(* LS Electric XG5000 project: 제일교회 *)
(* PLC LSPLC *)
(* module base 0 slot 0: Cnet:XGL-C42A/B (Cnet 통신 모듈(RS-422/485, RS-422/485)) *)
(* module base 0 slot 1: 입력 모듈:XGI-D24A/B (DC 24V 입력, 32점 (전류소스 싱크공용/ 전류소스 입력)) *)
(* module base 0 slot 2: 입력 모듈:XGI-D21A (DC 24V 입력, 8점 (전류소스/싱크입력)) *)
(* module base 0 slot 3: 출력 모듈:XGQ-TR4A/B (트랜지스터 출력, 32점 (0.1A용, 싱크출력/소스출력)) *)

(* Comments on direct variables
%MX100	MAIN POWER PBL
%MX101	십자가 PBL
%MX102	강대상 위 천정 PBL
%MX103	강대석(좌) PBL
%MX104	무대조명(좌) PBL
%MX105	(미정) PBL
%MX106	본당벽체 간접 PBL
%MX107	복도(좌) PBL
%MX108	중벽체(반달 좌) PBL
%MX109	중벽체 간접(좌) PBL
%MX110	기둥간접(좌) PBL
%MX111	중앙천정 강대상 PBL
%MX112	중앙천정앞(50W전구색) PBL
%MX113	중앙천정좌 간접 PBL
%MX114	중앙천정우 간접 PBL
%MX115	중앙천정U(20W주광색) PBL
%MX116	중앙천정뒤(50W전구색) PBL
%MX117	강대석 (우) PBL
%MX118	무대조명(우) PBL
%MX119	(미정) PBL
%MX120	본당벽체 간접 PBL
%MX121	복도(우) PBL
%MX122	중벽채(반달 우) PBL
%MX123	중벽체 간접(우) PBL
%MX124	기둥간접(우) PBL
%MX125	2층 후미 PBL
%MX126	종탑 PBL
%MX127	LAMP TEST PBL
%MX128	BUZZER STOP PBL[SR]
%MX129	RESET PBL[SR]
%MX130	SPARE
%MX131	SPARE
%MX200	MAIN POWER IN
%MX201	십자가 IN
%MX202	강대상 위 천정 IN
%MX203	강대석(좌) IN
%MX204	무대조명(좌) IN
%MX205	(미정) IN
%MX206	본당벽체 간접 IN
%MX207	복도 IN
%MX208	중벽체(반달) IN
%MX209	중벽체 간접 IN
%MX210	기둥간접 IN
%MX211	중앙천정 강대상 IN
%MX212	중앙천정앞(50W전구색) IN
%MX213	중앙천정좌 간접 IN
%MX214	중앙천정우 간접 IN
%MX215	중앙천정U(20W주광색) IN
%MX216	중앙천정뒤(50W전구색) IN
%MX217	강대석 (우) IN
%MX218	무대조명(우) IN
%MX219	(미정) IN
%MX220	본당벽체 간접 IN
%MX221	복도 IN
%MX222	중벽채(반달) IN
%MX223	중벽체 간접 IN
%MX224	기둥간접 IN
%MX225	2층 후미 IN
%MX226	종탑 IN
%MX227	LAMP TEST IN
%MX228	BUZZER STOP IN
%MX229	RESET IN
%MX230	SPARE IN
%MX231	SPARE IN
%MX300	MAIN POWER OUT
%MX301	십자가 OUT
%MX302	강대상 위 천정 OUT
%MX303	강대석(좌) OUT
%MX304	무대조명(좌) OUT
%MX305	(미정) OUT
%MX306	본당벽체 간접 OUT
%MX307	복도 OUT
%MX308	중벽체(반달) OUT
%MX309	중벽체 간접 OUT
%MX310	기둥간접 OUT
%MX311	중앙천정 강대상 OUT
%MX312	중앙천정앞(50W전구색) OUT
%MX313	중앙천정좌 간접 OUT
%MX314	중앙천정우 간접 OUT
%MX315	중앙천정U(20W주광색) OUT
%MX316	중앙천정뒤(50W전구색) OUT
%MX317	강대석 (우) OUT
%MX318	무대조명(우) OUT
%MX319	(미정) OUT
%MX320	본당벽체 간접 OUT
%MX321	복도 OUT
%MX322	중벽채(반달) OUT
%MX323	중벽체 간접 OUT
%MX324	기둥간접 OUT
%MX325	2층 후미 OUT
%MX326	종탑 OUT
%MX327	LAMP TEST OUT
%MX328	BUZZER STOP OUT
%MX329	RESET OUT
%MX330	SPARE OUT
%MX331	SPARE OUT
%MX400	MAIN POWER REMOTE
%MX401	십자가 REMOTE
%MX402	강대상 위 천정 REMOTE
%MX403	강대석(좌) REMOTE
%MX404	무대조명(좌) REMOTE
%MX405	(미정) REMOTE
%MX406	본당벽체 간접 REMOTE
%MX407	복도 REMOTE
%MX408	중벽체(반달) REMOTE
%MX409	중벽체 간접 REMOTE
%MX410	기둥간접 REMOTE
%MX411	중앙천정 강대상
REMOTE
%MX412	중앙천정앞
50W전구색
REMOTE
%MX413	중앙천정좌 간접 REMOTE
%MX414	중앙천정우 간접 REMOTE
%MX415	중앙천정U(20W주광색) REMOTE
%MX416	중앙천정뒤(50W전구색) REMOTE
%MX417	강대석 (우) REMOTE
%MX418	무대조명(우) REMOTE
%MX419	(미정) REMOTE
%MX420	본당벽체 간접 REMOTE
%MX421	복도 REMOTE
%MX422	중벽채(반달) REMOTE
%MX423	중벽체 간접 REMOTE
%MX424	기둥간접 REMOTE
%MX425	2층 후미 REMOTE
%MX426	종탑 REMOTE
%MX427	LAMP TEST REMOTE
%MX428	BUZZER STOP REMOTE
%MX429	RESET REMOTE
%MX430	SPARE REMOTE
%MX431	SPARE REMOTE
%MX500	MAIN POWER LAMP
%MX501	십자가 LAMP
%MX502	강대상 위 천정 LAMP
%MX503	강대석(좌) LAMP
%MX504	무대조명(좌) LAMP
%MX505	(미정) LAMP
%MX506	본당벽체 간접 LAMP
%MX507	복도 LAMP
%MX508	중벽체(반달) LAMP
%MX509	중벽체 간접 LAMP
%MX510	기둥간접 LAMP
%MX511	중앙천정 강대상 LAMP
%MX512	중앙천정앞(50W전구색) LAMP
%MX513	중앙천정좌 간접 LAMP
%MX514	중앙천정우 간접 LAMP
%MX515	중앙천정U(20W주광색) LAMP
%MX516	중앙천정뒤(50W전구색) LAMP
%MX517	강대석 (우) LAMP
%MX518	무대조명(우) LAMP
%MX519	(미정) LAMP
%MX520	본당벽체 간접 LAMP
%MX521	복도 LAMP
%MX522	중벽채(반달) LAMP
%MX523	중벽체 간접 LAMP
%MX524	기둥간접 LAMP
%MX525	2층 후미 LAMP
%MX526	종탑 LAMP
%MX527	LAMP TEST LAMP
%MX528	BUZZER STOP LAMP
%MX529	RESET LAMP
%MX530	BUZZER
[REMOTE]
%MX531	SPARE LAMP
%MX911	Total Alarm
%MX1000	중앙1열 S/W
%MX1001	중앙2열 S/W
%MX1002	중앙3열 S/W
%MX1003	중앙4열 S/W
%MX1004	중앙5열 S/W
%MX1005	중앙6열 S/W
%MX1006	중앙7열 S/W
%MX1007	중앙8열 S/W
%MX1008	중앙9열 S/W
%MX1009	중앙10열 S/W
%MX1010	장로석 S/W
%MX1011	장로석 SPOT S/W
%MX1012	성가대 S/W
%MX1013	성가대 SPOT S/W
%MX1014	좌측통로 S/W
%MX1015	우측통로 S/W
%MX1016	후단1열 S/W
%MX1017	후단2열 S/W
%MX1018	후단3열 S/W
%MX1019	종탑 
S/W
%MX1020	중앙1열 M/C-a
%MX1021	중앙2열 M/C-a
%MX1022	중앙3열 M/C-a
%MX1023	중앙4열 M/C-a
%MX1024	중앙5열 M/C-a
%MX1025	중앙6열 M/C-a
%MX1026	중앙7열 M/C-a
%MX1027	중앙8열 M/C-a
%MX1028	중앙9열 M/C-a
%MX1029	중앙10열 M/C-a
%MX1030	장로석 M/C-a
%MX1031	장로석 SPOT M/C-a
%MX1200	중앙1열 LOGIC
%MX1201	중앙2열 LOGIC
%MX1202	중앙3열 LOGIC
%MX1203	중앙4열 LOGIC
%MX1204	중앙5열 LOGIC
%MX1205	중앙6열 LOGIC
%MX1206	중앙7열 LOGIC
%MX1207	중앙8열 LOGIC
%MX1208	중앙9열 LOGIC
%MX1209	중앙10열 LOGIC
%MX1210	장로석 LOGIC
%MX1211	장로석 SPOT-LOGIC
%MX1212	성가대 LOGIC
%MX1213	성가대 SPOT-LOGIC
%MX1214	좌측통로 LOGIC
%MX1215	우측통로 LOGIC
%MX1216	후단1열 LOGIC
%MX1217	후단2열 LOGIC
%MX1218	후단3열 LOGIC
%MX1219	종탑 
LOGIC
%MX1220	중앙1열 M/C-a
%MX1221	중앙2열 M/C-a
%MX1222	중앙3열 M/C-a
%MX1223	중앙4열 M/C-a
%MX1224	중앙5열 M/C-a
%MX1225	중앙6열 M/C-a
%MX1226	중앙7열 M/C-a
%MX1227	중앙8열 M/C-a
%MX1228	중앙9열 M/C-a
%MX1229	중앙10열 M/C-a
%MX1230	장로석 M/C-a
%MX1231	장로석 SPOT M/C-a
%MX2000	성가대 M/C-a
%MX2001	성가대 SPOT M/C-a
%MX2002	좌측통로 M/C-a
%MX2003	우측통로 M/C-a
%MX2004	후단1열 M/C-a
%MX2005	후단2열 M/C-a
%MX2006	후단3열 M/C-a
%MX2007	종탑 
M/C-a
%MX2200	성가대 M/C-a
%MX2201	성가대 SPOT M/C-a
%MX2202	좌측통로 M/C-a
%MX2203	우측통로 M/C-a
%MX2204	후단1열 M/C-a
%MX2205	후단2열 M/C-a
%MX2206	후단3열 M/C-a
%MW0	IN-COM0
%MW1	IN-COM1
%MW2	OUT-COM0
%MW3	OUT-COM1
%IX0.1.0	중앙1열 S/W
%IX0.1.1	중앙2열 S/W
%IX0.1.2	중앙3열 S/W
%IX0.1.3	중앙4열 S/W
%IX0.1.4	중앙5열 S/W
%IX0.1.5	중앙6열 S/W
%IX0.1.6	중앙7열 S/W
%IX0.1.7	중앙8열 S/W
%IX0.1.8	중앙9열 S/W
%IX0.1.9	중앙10열 S/W
%IX0.1.10	장로석 S/W
%IX0.1.11	장로석 SPOT S/W
%IX0.1.12	성가대 S/W
%IX0.1.13	성가대 SPOT S/W
%IX0.1.14	좌측통로 S/W
%IX0.1.15	우측통로 S/W
%IX0.1.16	후단1열 S/W
%IX0.1.17	후단2열 S/W
%IX0.1.18	후단3열 S/W
%IX0.1.19	종탑
%IX0.1.20	중앙1열 M/C-a
%IX0.1.21	중앙2열 M/C-a
%IX0.1.22	중앙3열 M/C-a
%IX0.1.23	중앙4열 M/C-a
%IX0.1.24	중앙5열 M/C-a
%IX0.1.25	중앙6열 M/C-a
%IX0.1.26	중앙7열 M/C-a
%IX0.1.27	중앙8열 M/C-a
%IX0.1.28	중앙9열 M/C-a
%IX0.1.29	중앙10열 M/C-a
%IX0.1.30	장로석 M/C-a
%IX0.1.31	장로석 SPOT M/C-a
%IX0.2.0	성가대 M/C-a
%IX0.2.1	성가대 SPOT M/C-a
%IX0.2.2	좌측통로 M/C-a
%IX0.2.3	우측통로 M/C-a
%IX0.2.4	후단1열 M/C-a
%IX0.2.5	후단2열 M/C-a
%IX0.2.6	후단3열 M/C-a
%IX0.2.7	종탑
M/C-a
%QX0.3.0	중앙1열
%QX0.3.1	중앙2열
%QX0.3.2	중앙3열
%QX0.3.3	중앙4열
%QX0.3.4	중앙5열
%QX0.3.5	중앙6열
%QX0.3.6	중앙7열
%QX0.3.7	중앙8열
%QX0.3.8	중앙9열
%QX0.3.9	중앙10열
%QX0.3.10	장로석
%QX0.3.11	장로석 SPOT
%QX0.3.12	성가대
%QX0.3.13	성가대 SPOT
%QX0.3.14	좌측통로
%QX0.3.15	우측통로
%QX0.3.16	후단1열
%QX0.3.17	후단2열
%QX0.3.18	후단3열
%QX0.3.19	종탑
%QX0.3.20	BUZZER
[MAIN]
*)

PROGRAM Communication (* task: 스캔 프로그램 *)
VAR
    IN_0_HIGH : BYTE;
    IN_0_LOW : BYTE;
    IN_1_HIGH : BYTE;
    IN_1_LOW : BYTE;
    OUT_0_HIGH : BYTE;
    OUT_0_LOW : BYTE;
END_VAR

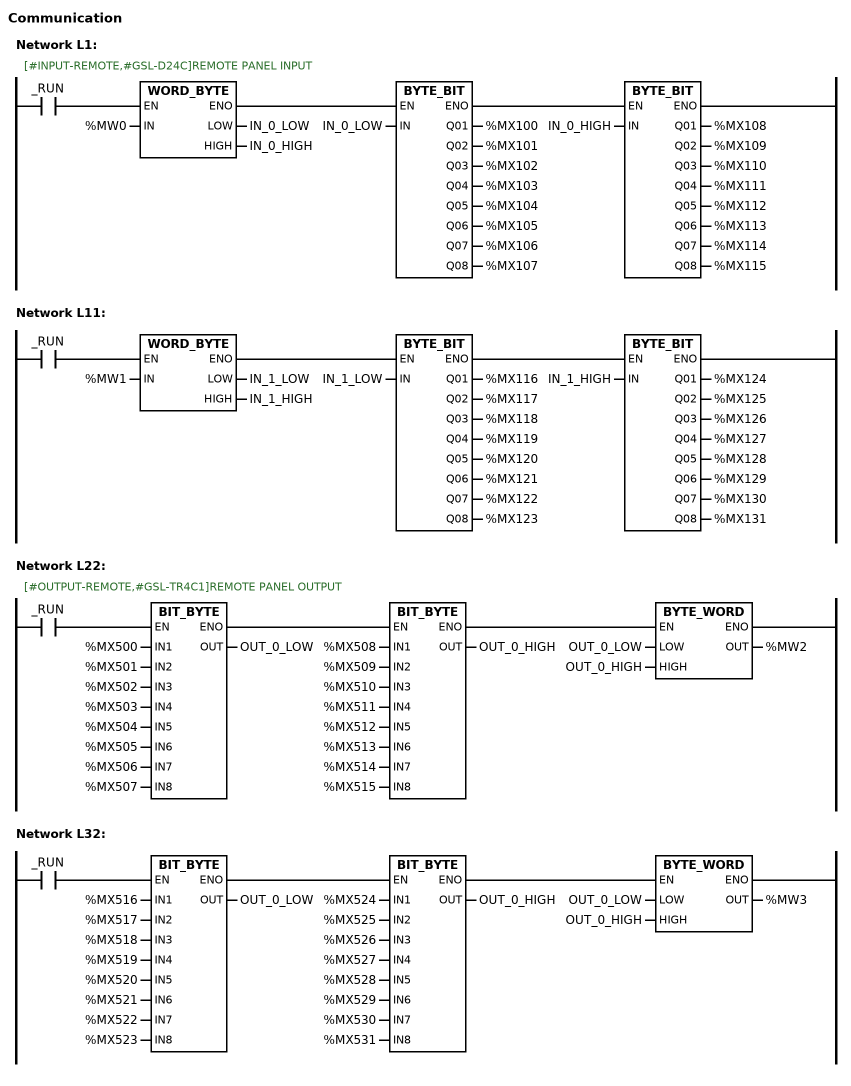
(* [#INPUT-REMOTE,#GSL-D24C]REMOTE PANEL INPUT *)
(* Rung L1 *)
IF _RUN THEN
    IN_0_LOW := WORD_BYTE(IN := %MW0, HIGH => IN_0_HIGH);
    %MX100 := BYTE_BIT(IN := IN_0_LOW, Q02 => %MX101, Q03 => %MX102, Q04 => %MX103, Q05 => %MX104, Q06 => %MX105, Q07 => %MX106, Q08 => %MX107);
    %MX108 := BYTE_BIT(IN := IN_0_HIGH, Q02 => %MX109, Q03 => %MX110, Q04 => %MX111, Q05 => %MX112, Q06 => %MX113, Q07 => %MX114, Q08 => %MX115);
END_IF;
(* Rung L11 *)
IF _RUN THEN
    IN_1_LOW := WORD_BYTE(IN := %MW1, HIGH => IN_1_HIGH);
    %MX116 := BYTE_BIT(IN := IN_1_LOW, Q02 => %MX117, Q03 => %MX118, Q04 => %MX119, Q05 => %MX120, Q06 => %MX121, Q07 => %MX122, Q08 => %MX123);
    %MX124 := BYTE_BIT(IN := IN_1_HIGH, Q02 => %MX125, Q03 => %MX126, Q04 => %MX127, Q05 => %MX128, Q06 => %MX129, Q07 => %MX130, Q08 => %MX131);
END_IF;
(* [#OUTPUT-REMOTE,#GSL-TR4C1]REMOTE PANEL OUTPUT *)
(* Rung L22 *)
IF _RUN THEN
    OUT_0_LOW := BIT_BYTE(%MX500, %MX501, %MX502, %MX503, %MX504, %MX505, %MX506, %MX507);
    OUT_0_HIGH := BIT_BYTE(%MX508, %MX509, %MX510, %MX511, %MX512, %MX513, %MX514, %MX515);
    %MW2 := BYTE_WORD(LOW := OUT_0_LOW, HIGH := OUT_0_HIGH);
END_IF;
(* Rung L32 *)
IF _RUN THEN
    OUT_0_LOW := BIT_BYTE(%MX516, %MX517, %MX518, %MX519, %MX520, %MX521, %MX522, %MX523);
    OUT_0_HIGH := BIT_BYTE(%MX524, %MX525, %MX526, %MX527, %MX528, %MX529, %MX530, %MX531);
    %MW3 := BYTE_WORD(LOW := OUT_0_LOW, HIGH := OUT_0_HIGH);
END_IF;
END_PROGRAM

PROGRAM Control-Remote (* task: 스캔 프로그램 *)
VAR
    FF0 : FF;
    FF1 : FF;
    FF10 : FF;
    FF11 : FF;
    FF12 : FF;
    FF13 : FF;
    FF14 : FF;
    FF15 : FF;
    FF16 : FF;
    FF17 : FF;
    FF18 : FF;
    FF19 : FF;
    FF2 : FF;
    FF20 : FF;
    FF21 : FF;
    FF22 : FF;
    FF23 : FF;
    FF24 : FF;
    FF25 : FF;
    FF26 : FF;
    FF27 : FF;
    FF28 : FF;
    FF29 : FF;
    FF3 : FF;
    FF30 : FF;
    FF31 : FF;
    FF4 : FF;
    FF5 : FF;
    FF6 : FF;
    FF7 : FF;
    FF8 : FF;
    FF9 : FF;
    INST : FF;
    INST1 : FF;
    IN_0_HIGH : BYTE;
    IN_0_LOW : BYTE;
    IN_1_HIGH : BYTE;
    IN_1_LOW : BYTE;
    off : BOOL;
END_VAR

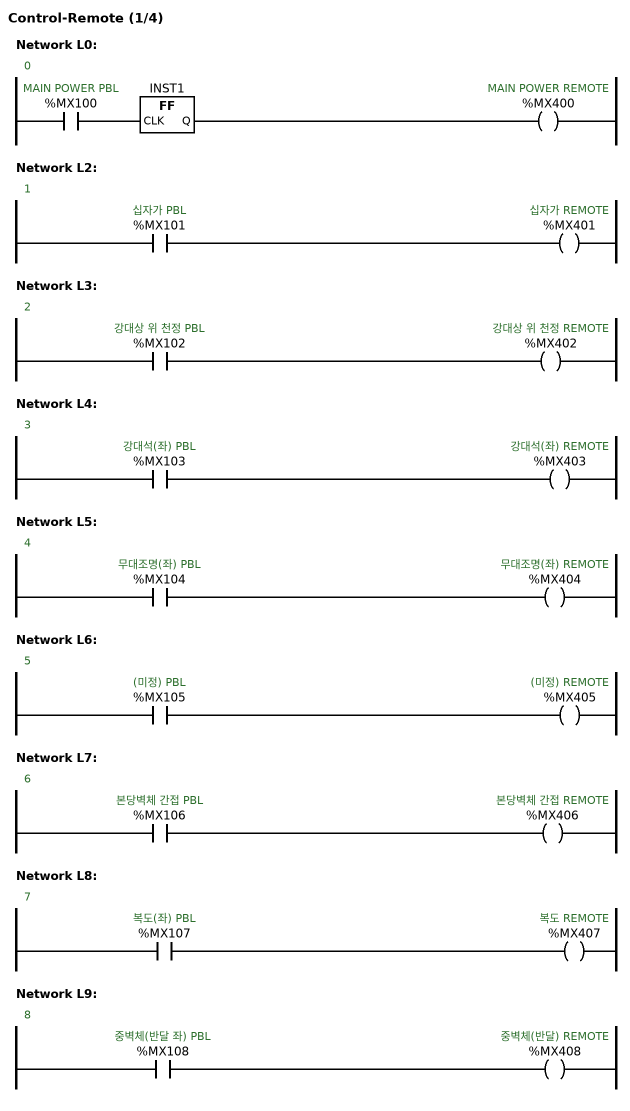
(* Rung L0 *)
INST1(CLK := %MX100);
%MX400 := INST1.Q;
(* 0 *)
(* Rung L2 *)
%MX401 := %MX101;
(* 1 *)
(* Rung L3 *)
%MX402 := %MX102;
(* 2 *)
(* Rung L4 *)
%MX403 := %MX103;
(* 3 *)
(* Rung L5 *)
%MX404 := %MX104;
(* 4 *)
(* Rung L6 *)
%MX405 := %MX105;
(* 5 *)
(* Rung L7 *)
%MX406 := %MX106;
(* 6 *)
(* Rung L8 *)
%MX407 := %MX107;
(* 7 *)
(* Rung L9 *)
%MX408 := %MX108;
(* 8 *)

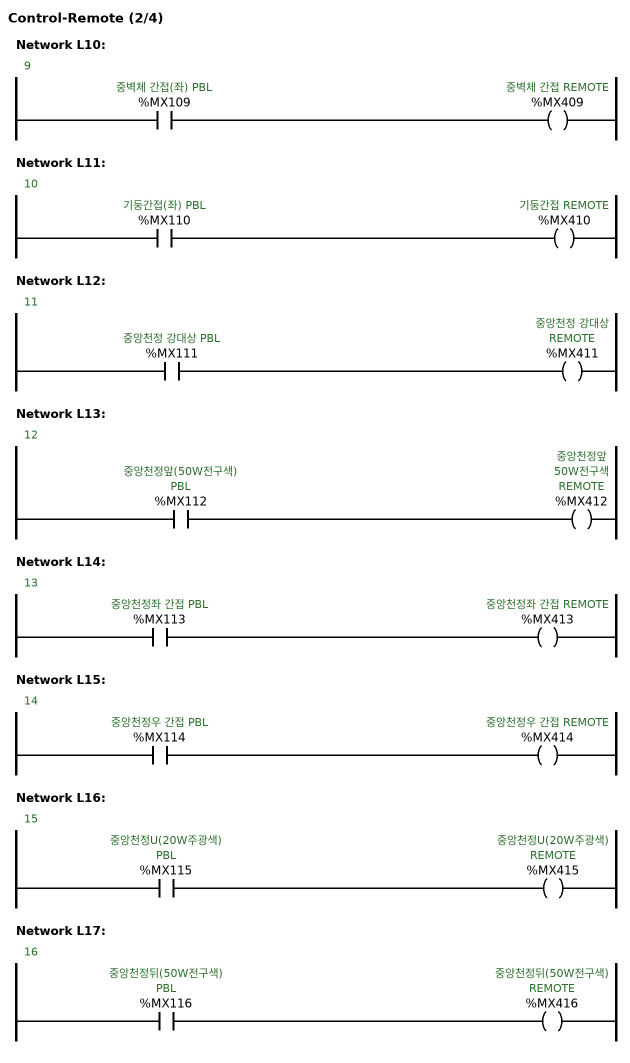
(* Rung L10 *)
%MX409 := %MX109;
(* 9 *)
(* Rung L11 *)
%MX410 := %MX110;
(* 10 *)
(* Rung L12 *)
%MX411 := %MX111;
(* 11 *)
(* Rung L13 *)
%MX412 := %MX112;
(* 12 *)
(* Rung L14 *)
%MX413 := %MX113;
(* 13 *)
(* Rung L15 *)
%MX414 := %MX114;
(* 14 *)
(* Rung L16 *)
%MX415 := %MX115;
(* 15 *)
(* Rung L17 *)
%MX416 := %MX116;
(* 16 *)

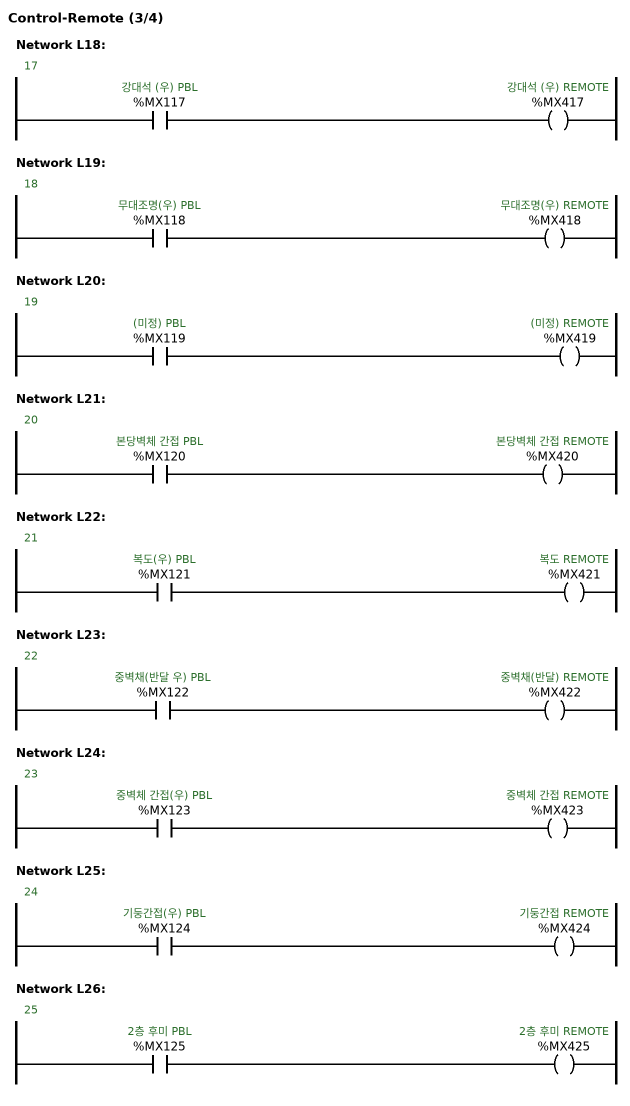
(* Rung L18 *)
%MX417 := %MX117;
(* 17 *)
(* Rung L19 *)
%MX418 := %MX118;
(* 18 *)
(* Rung L20 *)
%MX419 := %MX119;
(* 19 *)
(* Rung L21 *)
%MX420 := %MX120;
(* 20 *)
(* Rung L22 *)
%MX421 := %MX121;
(* 21 *)
(* Rung L23 *)
%MX422 := %MX122;
(* 22 *)
(* Rung L24 *)
%MX423 := %MX123;
(* 23 *)
(* Rung L25 *)
%MX424 := %MX124;
(* 24 *)
(* Rung L26 *)
%MX425 := %MX125;
(* 25 *)

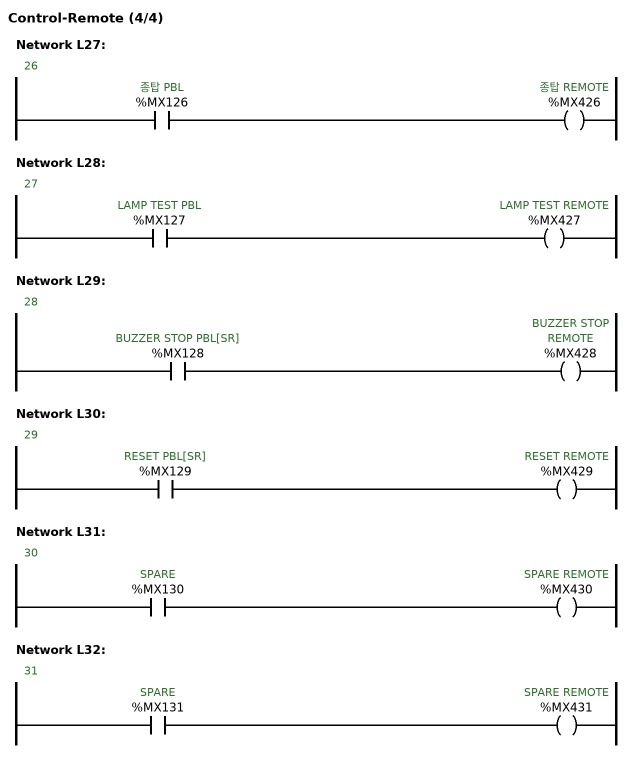
(* Rung L27 *)
%MX426 := %MX126;
(* 26 *)
(* Rung L28 *)
%MX427 := %MX127;
(* 27 *)
(* Rung L29 *)
%MX428 := %MX128;
(* 28 *)
(* Rung L30 *)
%MX429 := %MX129;
(* 29 *)
(* Rung L31 *)
%MX430 := %MX130;
(* 30 *)
(* Rung L32 *)
%MX431 := %MX131;
(* 31 *)
END_PROGRAM

PROGRAM Lamp-Remote (* task: 스캔 프로그램 *)
VAR
    INST : FF;
    INST1 : TMR_FLK;
    INST10 : TMR_FLK;
    INST2 : TMR_FLK;
    INST3 : TMR_FLK;
    INST4 : TMR_FLK;
    INST5 : TMR_FLK;
    INST6 : TMR_FLK;
    INST7 : TMR_FLK;
    INST8 : TMR_FLK;
    INST9 : TMR_FLK;
END_VAR

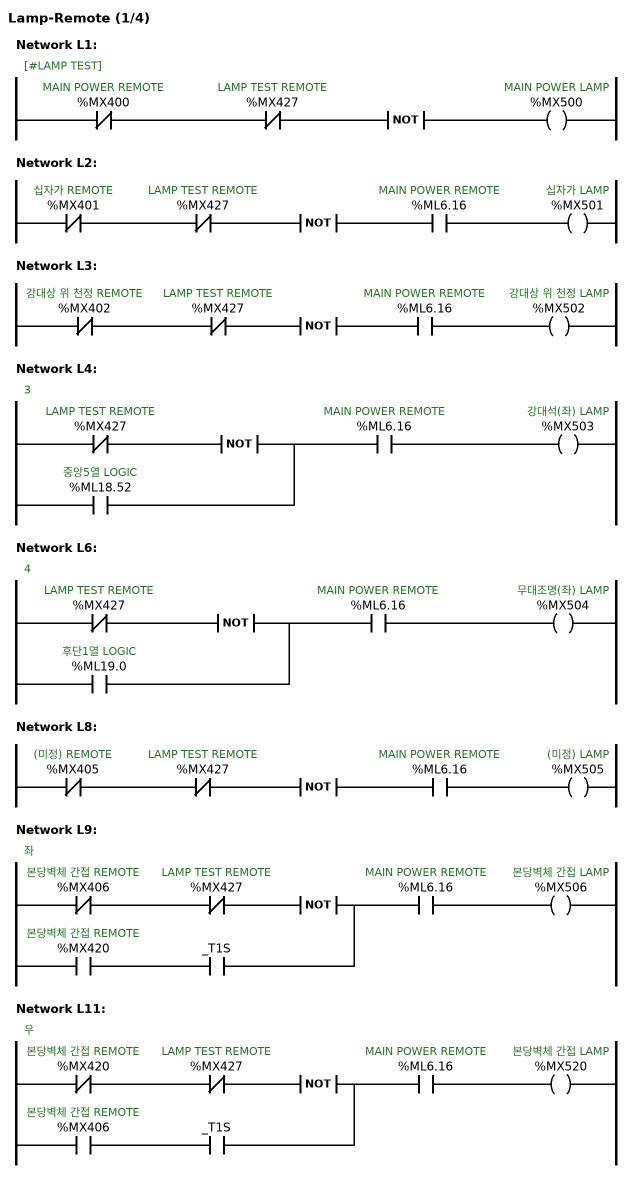
(* [#LAMP TEST] *)
(* Rung L1 *)
%MX500 := NOT (NOT %MX400 AND NOT %MX427);
(* Rung L2 *)
%MX501 := NOT (NOT %MX401 AND NOT %MX427) AND %ML6.16;
(* Rung L3 *)
%MX502 := NOT (NOT %MX402 AND NOT %MX427) AND %ML6.16;
(* Rung L4 *)
%MX503 := (%MX427 OR %ML18.52) AND %ML6.16;
(* 3 *)
(* Rung L6 *)
%MX504 := (%MX427 OR %ML19.0) AND %ML6.16;
(* 4 *)
(* Rung L8 *)
%MX505 := NOT (NOT %MX405 AND NOT %MX427) AND %ML6.16;
(* Rung L9 *)
%MX506 := (NOT (NOT %MX406 AND NOT %MX427) OR (%MX420 AND _T1S)) AND %ML6.16;
(* 좌 *)
(* Rung L11 *)
%MX520 := (NOT (NOT %MX420 AND NOT %MX427) OR (%MX406 AND _T1S)) AND %ML6.16;
(* 우 *)

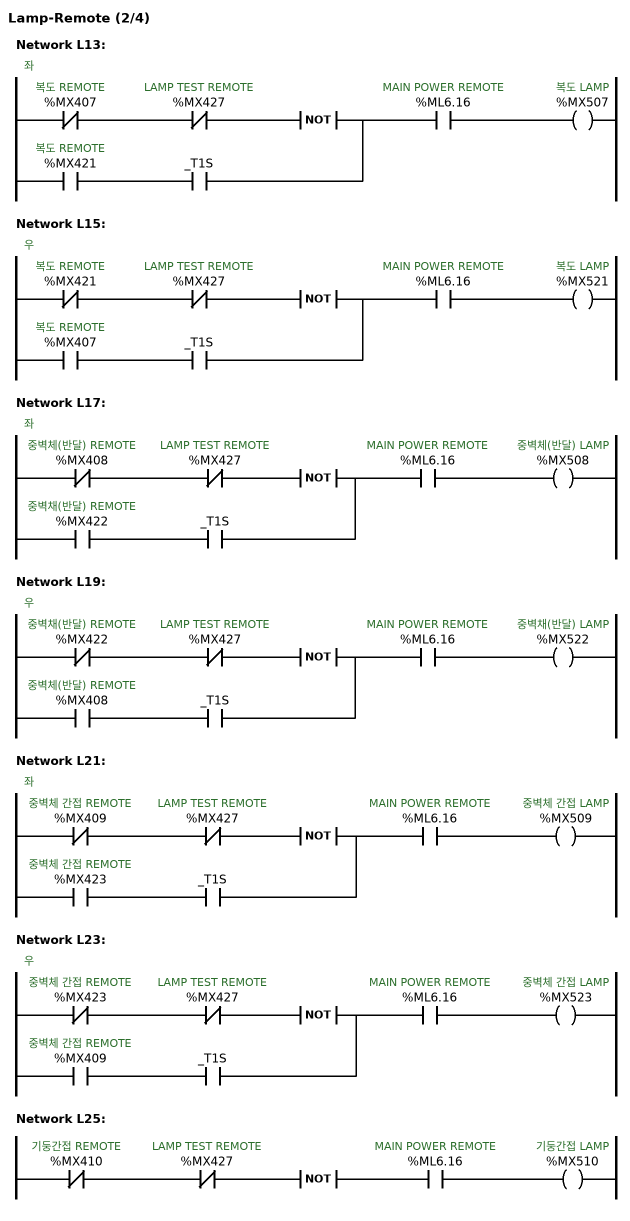
(* Rung L13 *)
%MX507 := (NOT (NOT %MX407 AND NOT %MX427) OR (%MX421 AND _T1S)) AND %ML6.16;
(* 좌 *)
(* Rung L15 *)
%MX521 := (NOT (NOT %MX421 AND NOT %MX427) OR (%MX407 AND _T1S)) AND %ML6.16;
(* 우 *)
(* Rung L17 *)
%MX508 := (NOT (NOT %MX408 AND NOT %MX427) OR (%MX422 AND _T1S)) AND %ML6.16;
(* 좌 *)
(* Rung L19 *)
%MX522 := (NOT (NOT %MX422 AND NOT %MX427) OR (%MX408 AND _T1S)) AND %ML6.16;
(* 우 *)
(* Rung L21 *)
%MX509 := (NOT (NOT %MX409 AND NOT %MX427) OR (%MX423 AND _T1S)) AND %ML6.16;
(* 좌 *)
(* Rung L23 *)
%MX523 := (NOT (NOT %MX423 AND NOT %MX427) OR (%MX409 AND _T1S)) AND %ML6.16;
(* 우 *)
(* Rung L25 *)
%MX510 := NOT (NOT %MX410 AND NOT %MX427) AND %ML6.16;

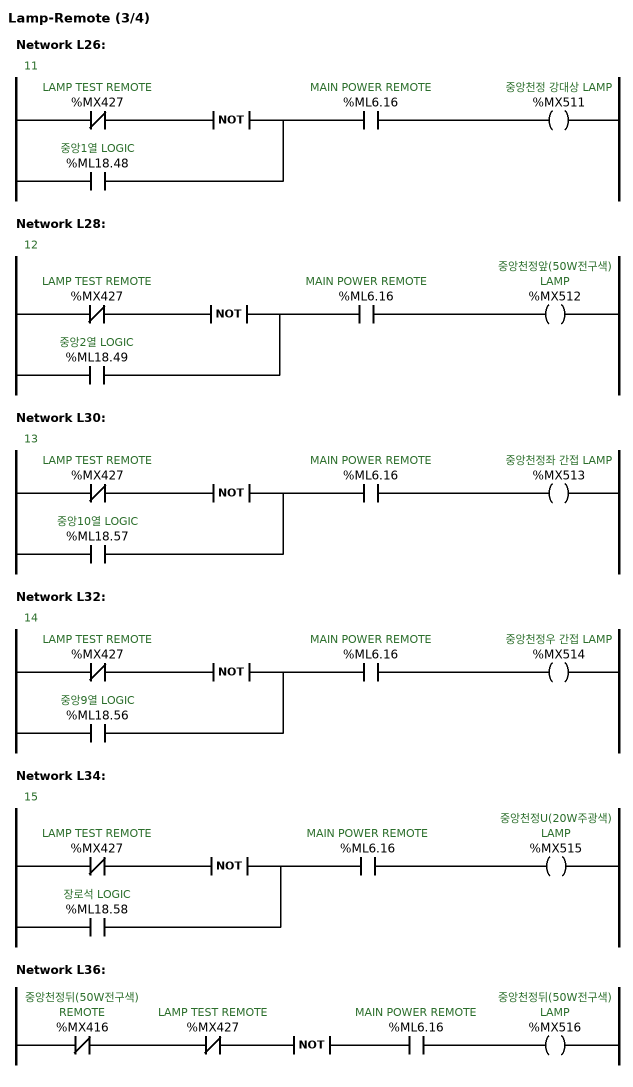
(* Rung L26 *)
%MX511 := (%MX427 OR %ML18.48) AND %ML6.16;
(* 11 *)
(* Rung L28 *)
%MX512 := (%MX427 OR %ML18.49) AND %ML6.16;
(* 12 *)
(* Rung L30 *)
%MX513 := (%MX427 OR %ML18.57) AND %ML6.16;
(* 13 *)
(* Rung L32 *)
%MX514 := (%MX427 OR %ML18.56) AND %ML6.16;
(* 14 *)
(* Rung L34 *)
%MX515 := (%MX427 OR %ML18.58) AND %ML6.16;
(* 15 *)
(* Rung L36 *)
%MX516 := NOT (NOT %MX416 AND NOT %MX427) AND %ML6.16;

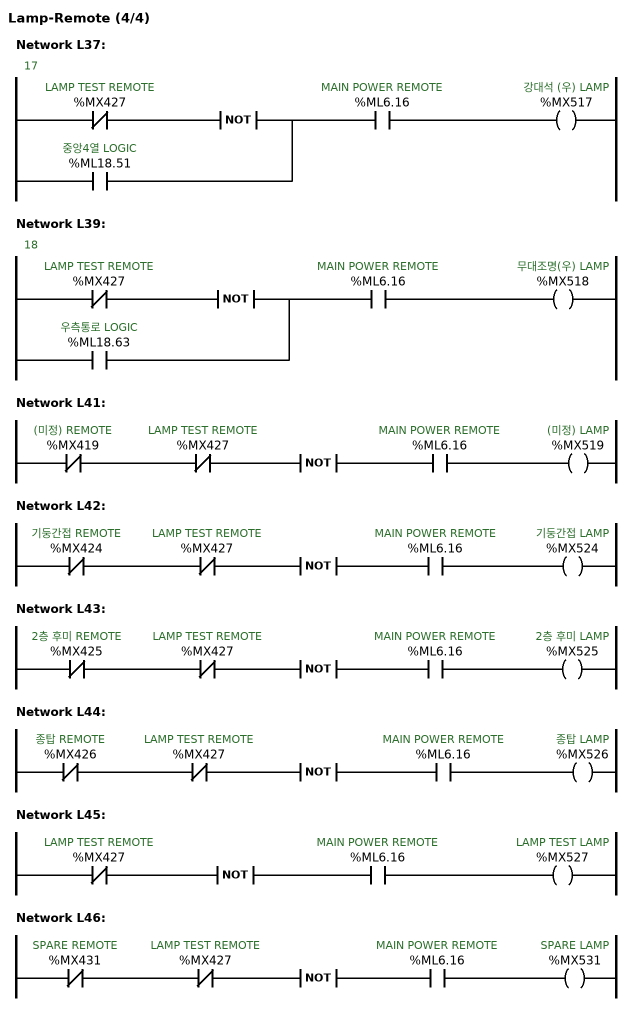
(* Rung L37 *)
%MX517 := (%MX427 OR %ML18.51) AND %ML6.16;
(* 17 *)
(* Rung L39 *)
%MX518 := (%MX427 OR %ML18.63) AND %ML6.16;
(* 18 *)
(* Rung L41 *)
%MX519 := NOT (NOT %MX419 AND NOT %MX427) AND %ML6.16;
(* Rung L42 *)
%MX524 := NOT (NOT %MX424 AND NOT %MX427) AND %ML6.16;
(* Rung L43 *)
%MX525 := NOT (NOT %MX425 AND NOT %MX427) AND %ML6.16;
(* Rung L44 *)
%MX526 := NOT (NOT %MX426 AND NOT %MX427) AND %ML6.16;
(* Rung L45 *)
%MX527 := %MX427 AND %ML6.16;
(* Rung L46 *)
%MX531 := NOT (NOT %MX431 AND NOT %MX427) AND %ML6.16;
END_PROGRAM

PROGRAM INPUT-MAIN (* task: 스캔 프로그램 *)

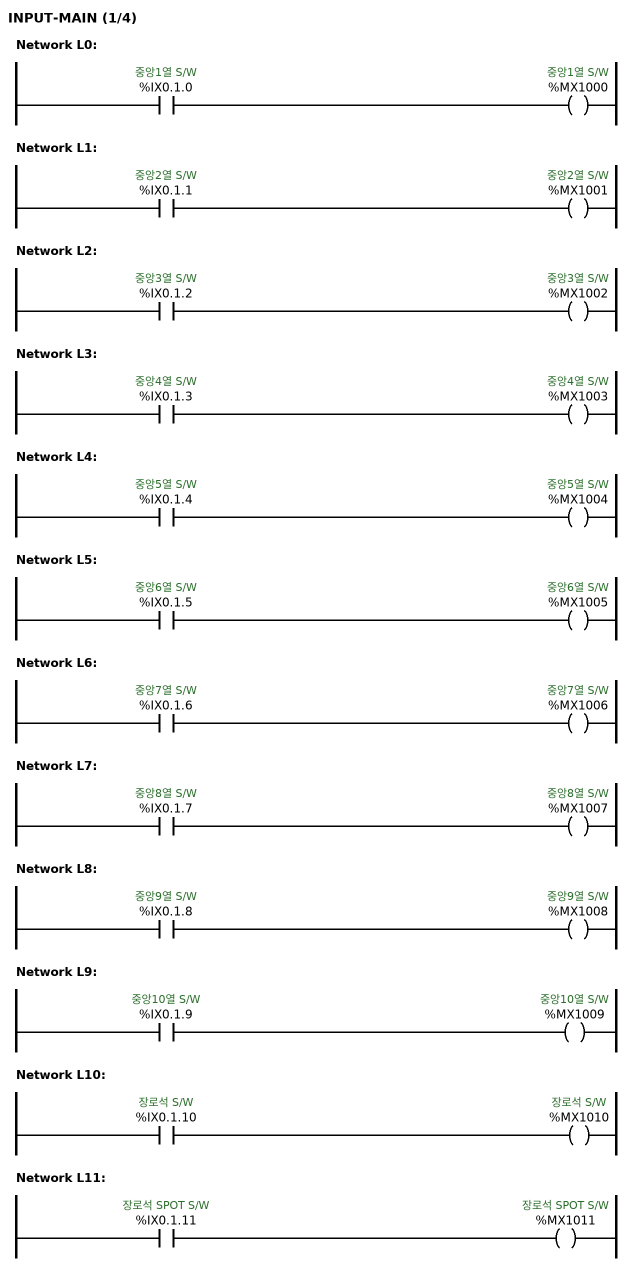
(* Rung L0 *)
%MX1000 := %IX0.1.0;
(* Rung L1 *)
%MX1001 := %IX0.1.1;
(* Rung L2 *)
%MX1002 := %IX0.1.2;
(* Rung L3 *)
%MX1003 := %IX0.1.3;
(* Rung L4 *)
%MX1004 := %IX0.1.4;
(* Rung L5 *)
%MX1005 := %IX0.1.5;
(* Rung L6 *)
%MX1006 := %IX0.1.6;
(* Rung L7 *)
%MX1007 := %IX0.1.7;
(* Rung L8 *)
%MX1008 := %IX0.1.8;
(* Rung L9 *)
%MX1009 := %IX0.1.9;
(* Rung L10 *)
%MX1010 := %IX0.1.10;
(* Rung L11 *)
%MX1011 := %IX0.1.11;

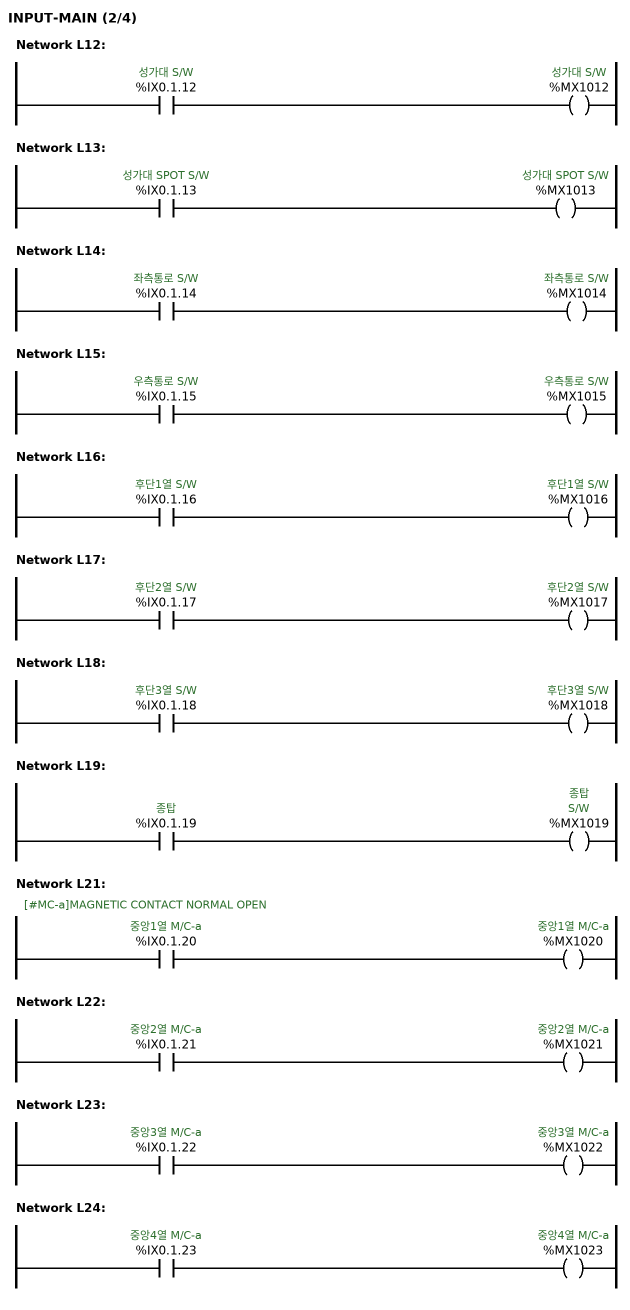
(* Rung L12 *)
%MX1012 := %IX0.1.12;
(* Rung L13 *)
%MX1013 := %IX0.1.13;
(* Rung L14 *)
%MX1014 := %IX0.1.14;
(* Rung L15 *)
%MX1015 := %IX0.1.15;
(* Rung L16 *)
%MX1016 := %IX0.1.16;
(* Rung L17 *)
%MX1017 := %IX0.1.17;
(* Rung L18 *)
%MX1018 := %IX0.1.18;
(* Rung L19 *)
%MX1019 := %IX0.1.19;
(* [#MC-a]MAGNETIC CONTACT NORMAL OPEN *)
(* Rung L21 *)
%MX1020 := %IX0.1.20;
(* Rung L22 *)
%MX1021 := %IX0.1.21;
(* Rung L23 *)
%MX1022 := %IX0.1.22;
(* Rung L24 *)
%MX1023 := %IX0.1.23;

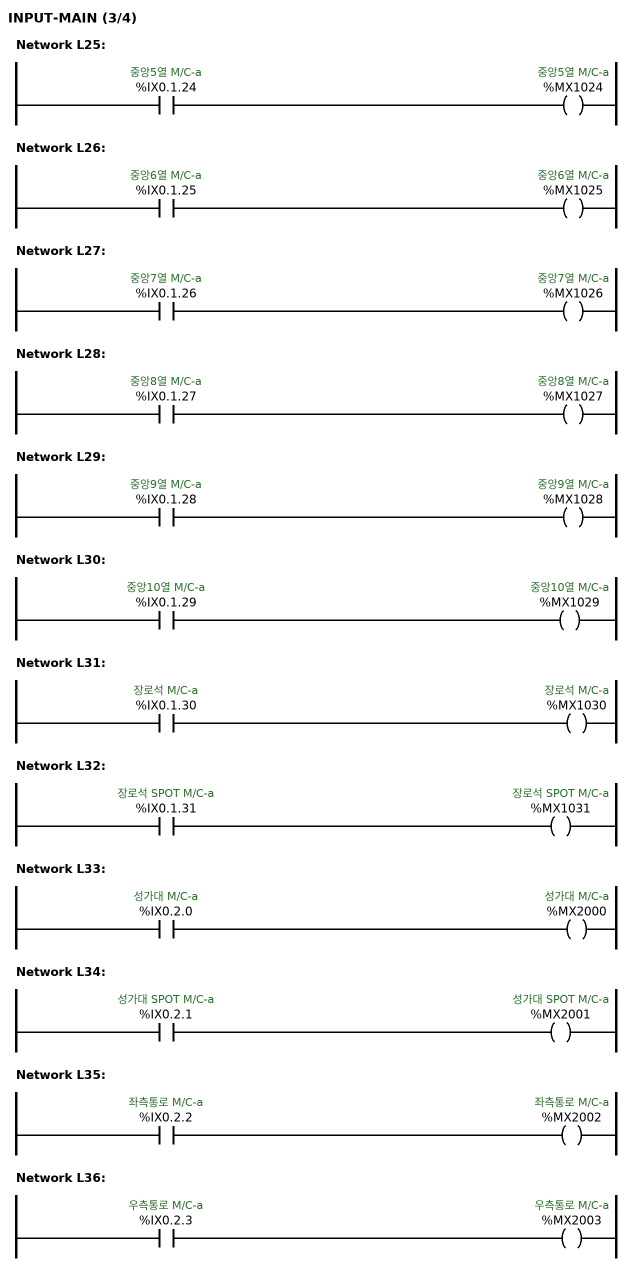
(* Rung L25 *)
%MX1024 := %IX0.1.24;
(* Rung L26 *)
%MX1025 := %IX0.1.25;
(* Rung L27 *)
%MX1026 := %IX0.1.26;
(* Rung L28 *)
%MX1027 := %IX0.1.27;
(* Rung L29 *)
%MX1028 := %IX0.1.28;
(* Rung L30 *)
%MX1029 := %IX0.1.29;
(* Rung L31 *)
%MX1030 := %IX0.1.30;
(* Rung L32 *)
%MX1031 := %IX0.1.31;
(* Rung L33 *)
%MX2000 := %IX0.2.0;
(* Rung L34 *)
%MX2001 := %IX0.2.1;
(* Rung L35 *)
%MX2002 := %IX0.2.2;
(* Rung L36 *)
%MX2003 := %IX0.2.3;

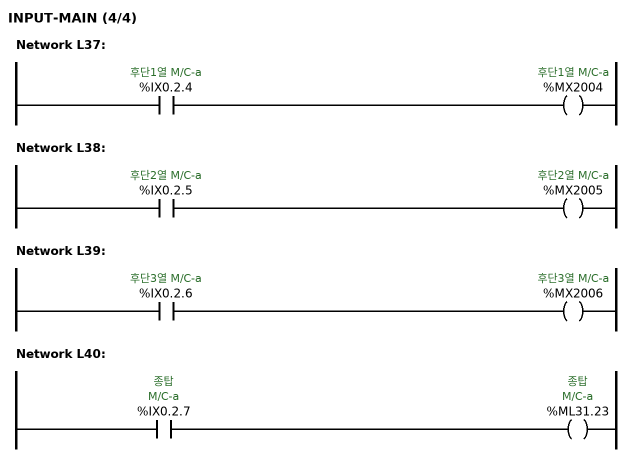
(* Rung L37 *)
%MX2004 := %IX0.2.4;
(* Rung L38 *)
%MX2005 := %IX0.2.5;
(* Rung L39 *)
%MX2006 := %IX0.2.6;
(* Rung L40 *)
%ML31.23 := %IX0.2.7;
END_PROGRAM

PROGRAM LAMP-CONTROL (* task: 스캔 프로그램 *)
VAR
    INST : FF;
    INST1 : FF;
    INST10 : FF;
    INST2 : FF;
    INST3 : FF;
    INST4 : FF;
    INST5 : FF;
    INST6 : FF;
    INST7 : FF;
    INST8 : FF;
    INST9 : FF;
END_VAR

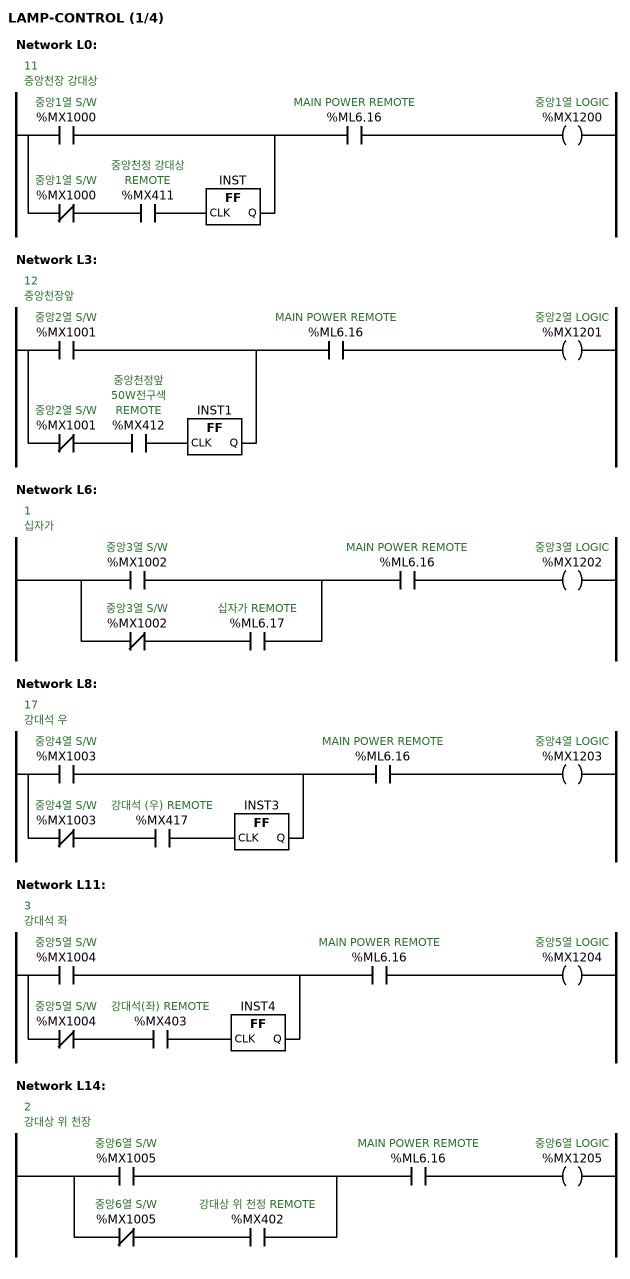
(* Rung L0 *)
INST(CLK := NOT %MX1000 AND %MX411);
%MX1200 := (%MX1000 OR INST.Q) AND %ML6.16;
(* 11 / 중앙천장 강대상 *)
(* Rung L3 *)
INST1(CLK := NOT %MX1001 AND %MX412);
%MX1201 := (%MX1001 OR INST1.Q) AND %ML6.16;
(* 12 / 중앙천장앞 *)
(* Rung L6 *)
%MX1202 := (%MX1002 OR (NOT %MX1002 AND %ML6.17)) AND %ML6.16;
(* 1 / 십자가 *)
(* Rung L8 *)
INST3(CLK := NOT %MX1003 AND %MX417);
%MX1203 := (%MX1003 OR INST3.Q) AND %ML6.16;
(* 17 / 강대석 우 *)
(* Rung L11 *)
INST4(CLK := NOT %MX1004 AND %MX403);
%MX1204 := (%MX1004 OR INST4.Q) AND %ML6.16;
(* 3 / 강대석 좌 *)
(* Rung L14 *)
%MX1205 := (%MX1005 OR (NOT %MX1005 AND %MX402)) AND %ML6.16;
(* 2 / 강대상 위 천장 *)

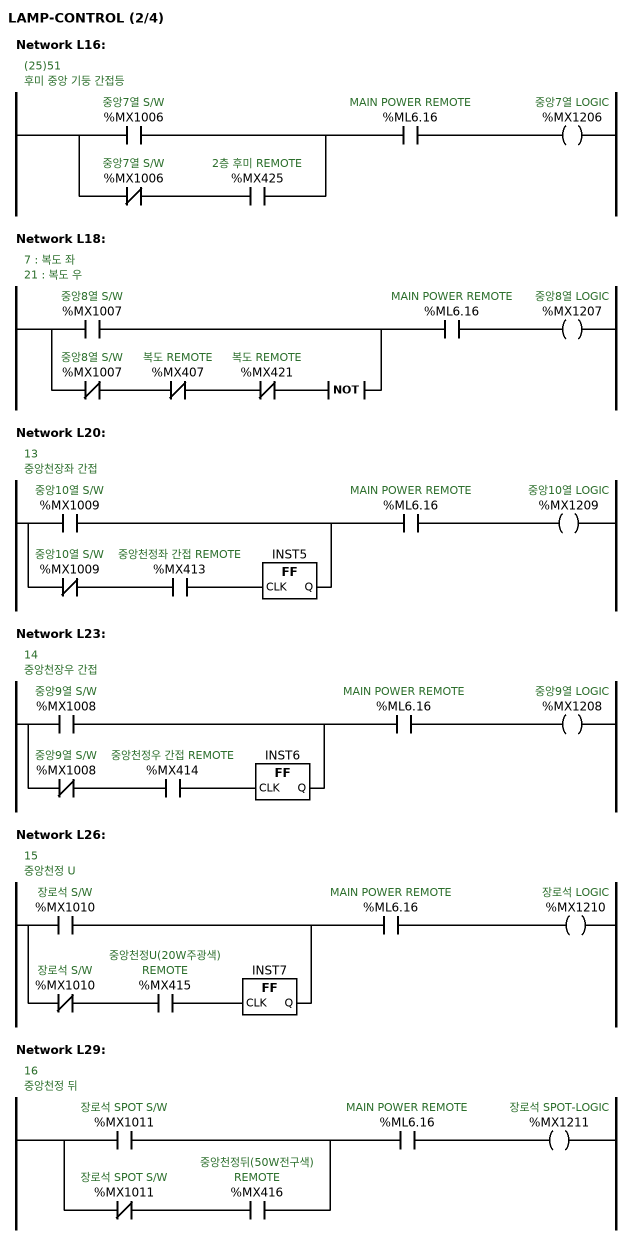
(* Rung L16 *)
%MX1206 := (%MX1006 OR (NOT %MX1006 AND %MX425)) AND %ML6.16;
(* (25)51 / 후미 중앙 기둥 간접등 *)
(* Rung L18 *)
%MX1207 := (%MX1007 OR NOT (NOT %MX1007 AND NOT %MX407 AND NOT %MX421)) AND %ML6.16;
(* 7 : 복도 좌 / 21 : 복도 우 *)
(* Rung L20 *)
INST5(CLK := NOT %MX1009 AND %MX413);
%MX1209 := (%MX1009 OR INST5.Q) AND %ML6.16;
(* 13 / 중앙천장좌 간접 *)
(* Rung L23 *)
INST6(CLK := NOT %MX1008 AND %MX414);
%MX1208 := (%MX1008 OR INST6.Q) AND %ML6.16;
(* 14 / 중앙천장우 간접 *)
(* Rung L26 *)
INST7(CLK := NOT %MX1010 AND %MX415);
%MX1210 := (%MX1010 OR INST7.Q) AND %ML6.16;
(* 15 / 중앙천정 U *)
(* Rung L29 *)
%MX1211 := (%MX1011 OR (NOT %MX1011 AND %MX416)) AND %ML6.16;
(* 16 / 중앙천정 뒤 *)

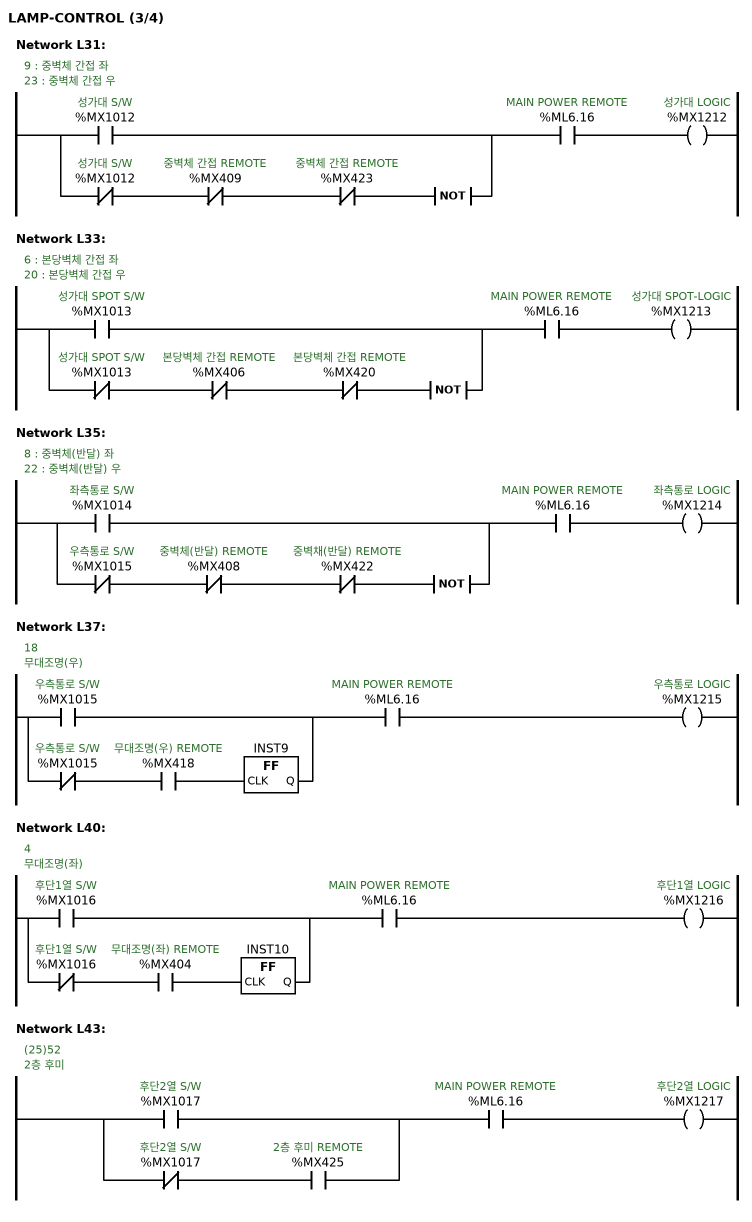
(* Rung L31 *)
%MX1212 := (%MX1012 OR NOT (NOT %MX1012 AND NOT %MX409 AND NOT %MX423)) AND %ML6.16;
(* 9 : 중벽체 간접 좌 / 23 : 중벽체 간접 우 *)
(* Rung L33 *)
%MX1213 := (%MX1013 OR NOT (NOT %MX1013 AND NOT %MX406 AND NOT %MX420)) AND %ML6.16;
(* 6 : 본당벽체 간접 좌 / 20 : 본당벽체 간접 우 *)
(* Rung L35 *)
%MX1214 := (%MX1014 OR NOT (NOT %MX1015 AND NOT %MX408 AND NOT %MX422)) AND %ML6.16;
(* 8 : 중벽체(반달) 좌 / 22 : 중벽체(반달) 우 *)
(* Rung L37 *)
INST9(CLK := NOT %MX1015 AND %MX418);
%MX1215 := (%MX1015 OR INST9.Q) AND %ML6.16;
(* 18 / 무대조명(우) *)
(* Rung L40 *)
INST10(CLK := NOT %MX1016 AND %MX404);
%MX1216 := (%MX1016 OR INST10.Q) AND %ML6.16;
(* 4 / 무대조명(좌) *)
(* Rung L43 *)
%MX1217 := (%MX1017 OR (NOT %MX1017 AND %MX425)) AND %ML6.16;
(* (25)52 / 2층 후미 *)

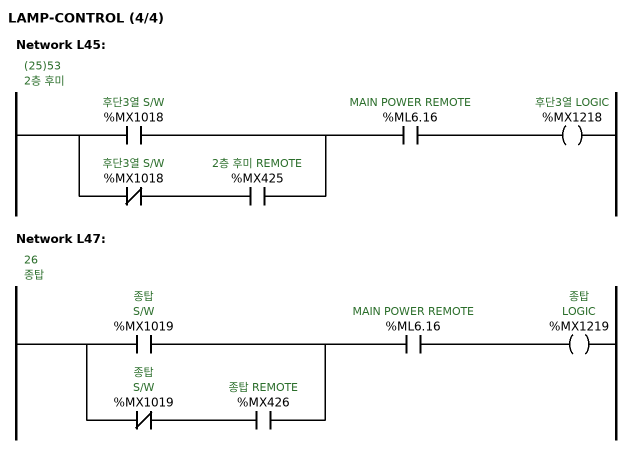
(* Rung L45 *)
%MX1218 := (%MX1018 OR (NOT %MX1018 AND %MX425)) AND %ML6.16;
(* (25)53 / 2층 후미 *)
(* Rung L47 *)
%MX1219 := (%MX1019 OR (NOT %MX1019 AND %MX426)) AND %ML6.16;
(* 26 / 종탑 *)
END_PROGRAM

PROGRAM OUTPUT-MAIN (* task: 스캔 프로그램 *)

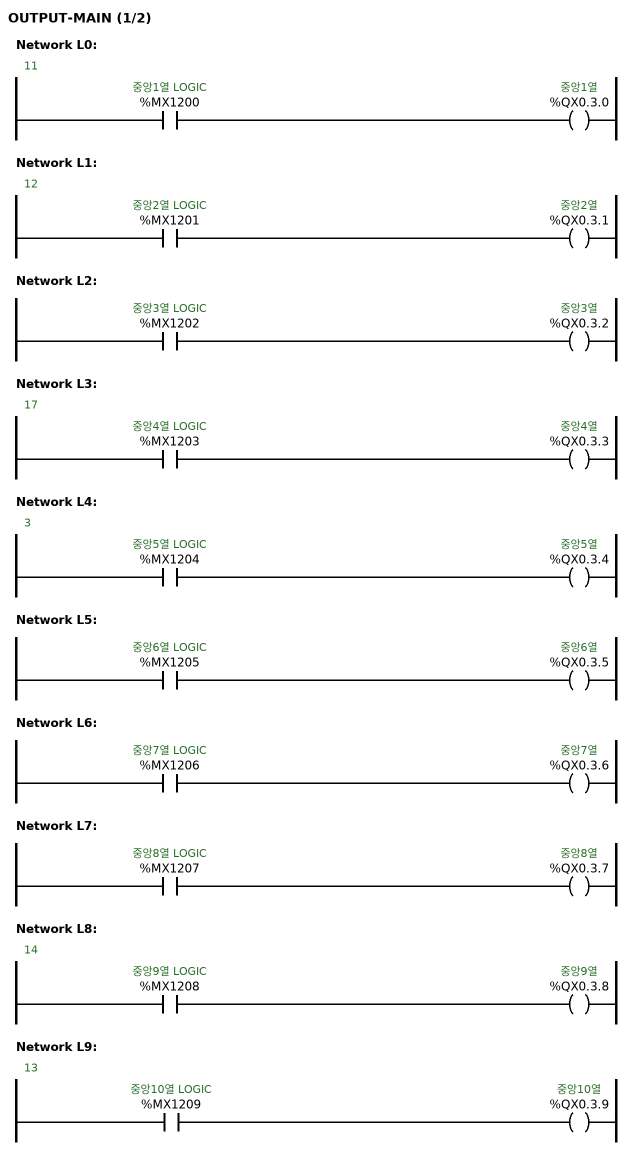
(* Rung L0 *)
%QX0.3.0 := %MX1200;
(* 11 *)
(* Rung L1 *)
%QX0.3.1 := %MX1201;
(* 12 *)
(* Rung L2 *)
%QX0.3.2 := %MX1202;
(* Rung L3 *)
%QX0.3.3 := %MX1203;
(* 17 *)
(* Rung L4 *)
%QX0.3.4 := %MX1204;
(* 3 *)
(* Rung L5 *)
%QX0.3.5 := %MX1205;
(* Rung L6 *)
%QX0.3.6 := %MX1206;
(* Rung L7 *)
%QX0.3.7 := %MX1207;
(* Rung L8 *)
%QX0.3.8 := %MX1208;
(* 14 *)
(* Rung L9 *)
%QX0.3.9 := %MX1209;
(* 13 *)

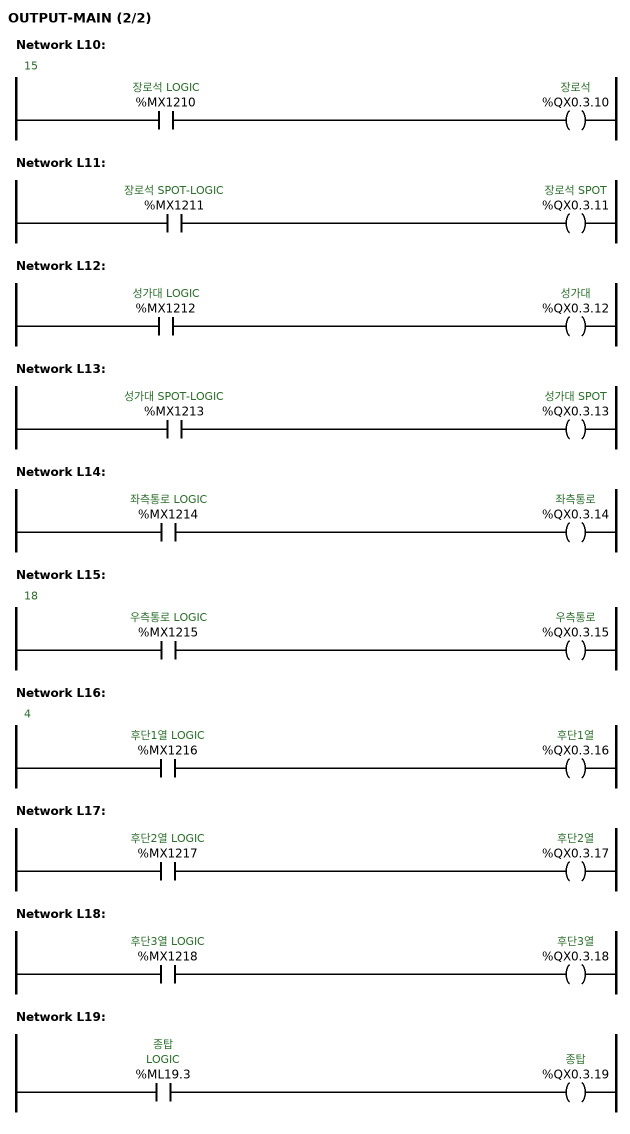
(* Rung L10 *)
%QX0.3.10 := %MX1210;
(* 15 *)
(* Rung L11 *)
%QX0.3.11 := %MX1211;
(* Rung L12 *)
%QX0.3.12 := %MX1212;
(* Rung L13 *)
%QX0.3.13 := %MX1213;
(* Rung L14 *)
%QX0.3.14 := %MX1214;
(* Rung L15 *)
%QX0.3.15 := %MX1215;
(* 18 *)
(* Rung L16 *)
%QX0.3.16 := %MX1216;
(* 4 *)
(* Rung L17 *)
%QX0.3.17 := %MX1217;
(* Rung L18 *)
%QX0.3.18 := %MX1218;
(* Rung L19 *)
%QX0.3.19 := %ML19.3;
END_PROGRAM

PROGRAM ALARM (* task: 스캔 프로그램 *)
VAR
    BUZZER : BOOL; (* BUZZER / SIG *)
    BZ_STOP : BOOL;
    FF : FF;
    INST : FF;
    INST1 : FF;
    INST2 : TON;
    INST9 : TMR_FLK;
END_VAR
VAR
    _p1 : BOOL;
    _p2 : BOOL;
END_VAR

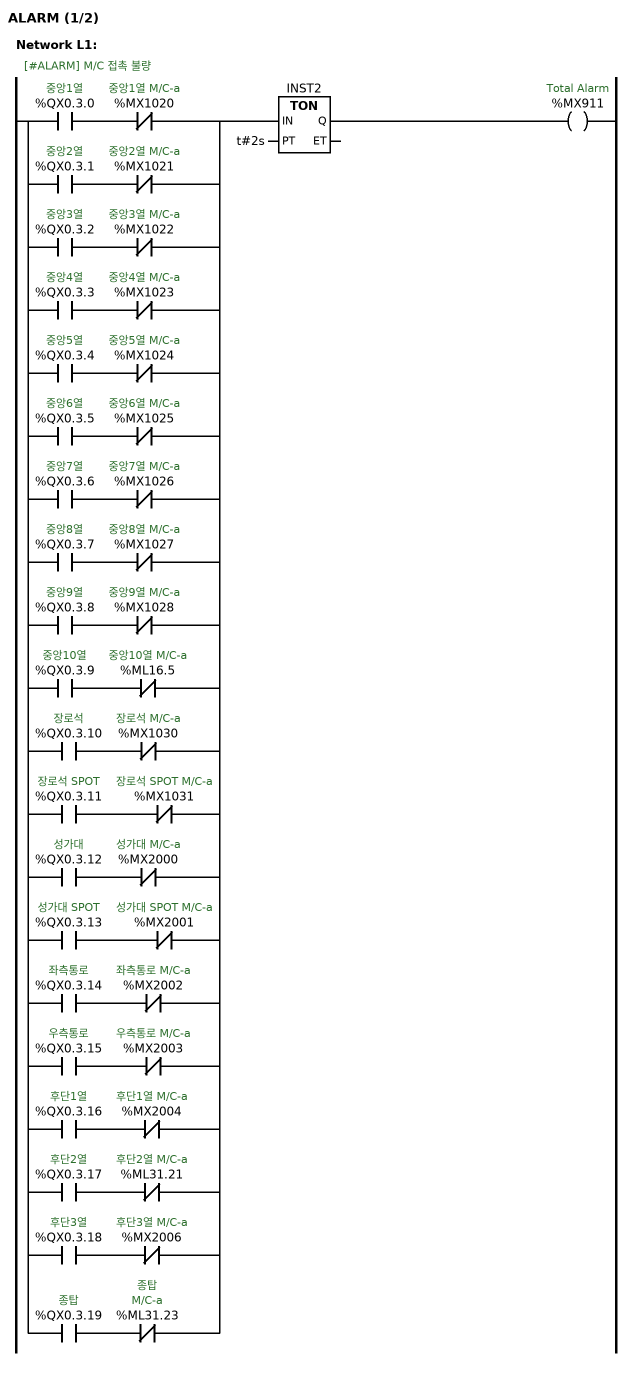
(* [#ALARM] M/C 접촉 불량 *)
(* Rung L1 *)
INST2(IN := (%QX0.3.0 AND NOT %MX1020) OR (%QX0.3.1 AND NOT %MX1021) OR (%QX0.3.2 AND NOT %MX1022) OR (%QX0.3.3 AND NOT %MX1023) OR (%QX0.3.4 AND NOT %MX1024) OR (%QX0.3.5 AND NOT %MX1025) OR (%QX0.3.6 AND NOT %MX1026) OR (%QX0.3.7 AND NOT %MX1027) OR (%QX0.3.8 AND NOT %MX1028) OR (%QX0.3.9 AND NOT %ML16.5) OR (%QX0.3.10 AND NOT %MX1030) OR (%QX0.3.11 AND NOT %MX1031) OR (%QX0.3.12 AND NOT %MX2000) OR (%QX0.3.13 AND NOT %MX2001) OR (%QX0.3.14 AND NOT %MX2002) OR (%QX0.3.15 AND NOT %MX2003) OR (%QX0.3.16 AND NOT %MX2004) OR (%QX0.3.17 AND NOT %ML31.21) OR (%QX0.3.18 AND NOT %MX2006) OR (%QX0.3.19 AND NOT %ML31.23), PT := t#2s);
%MX911 := INST2.Q;

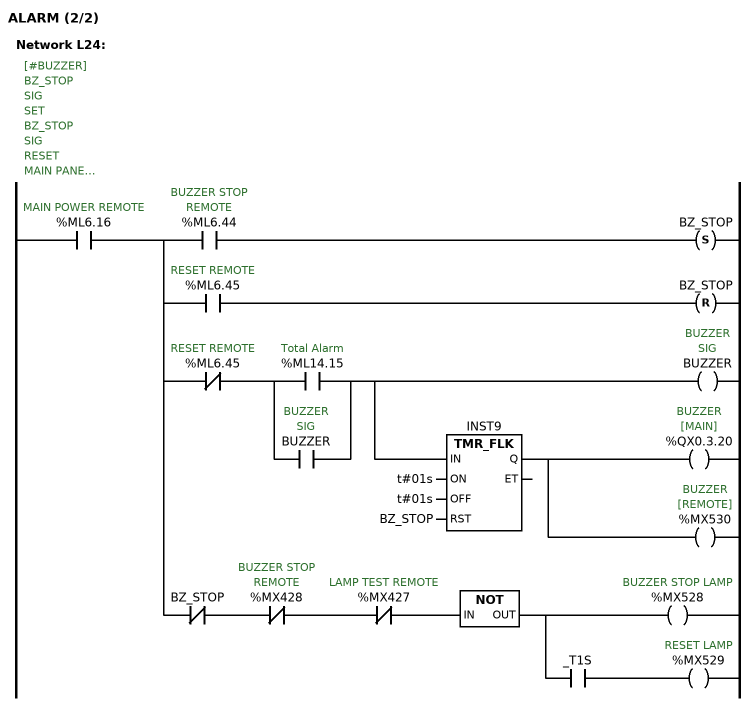
(* [#BUZZER] *)
(* Rung L24 *)
IF %ML6.16 AND %ML6.44 THEN BZ_STOP := TRUE; END_IF;
IF %ML6.16 AND %ML6.45 THEN BZ_STOP := FALSE; END_IF;
_p1 := %ML6.16 AND NOT %ML6.45 AND (%ML14.15 OR BUZZER);
BUZZER := _p1;
INST9(IN := _p1, ON := t#01s, OFF := t#01s, RST := BZ_STOP);
%QX0.3.20 := INST9.Q;
%MX530 := INST9.Q;
_p2 := NOT (%ML6.16 AND NOT BZ_STOP AND NOT %MX428 AND NOT %MX427);
%MX528 := _p2;
%MX529 := _p2 AND _T1S;
(* BZ_STOP / SIG / SET *)
(* BZ_STOP / SIG / RESET *)
(* MAIN PANEL / BUZZER / OUTPUT *)
(* REMOTE PANEL / BUZZER / OUTPUT *)
END_PROGRAM